{attribute 'qualified_only'}
{attribute 'strict'}
{attribute 'to_string'}
TYPE eTcaCarrierCmd :
(
	noCmd := 0,
	emptyPlaces,
	fillPlaces,
	RestorePlaces,
	ConfigCarrier
);
END_TYPE

(* stored: Version 1.1.0.1
   DUT eTcaCarrierCmd: Id {1e38e4ae-ea61-4cf0-bd3f-f87d1f3b8ecf} *)
